DATA_BLOCK "KukaRobot2_CtrlDB"
{ S7_Optimized_Access := 'FALSE' }
VERSION : 0.1
"KukaRobot2_Ctrl"

BEGIN

END_DATA_BLOCK

